(* IEC 61131-3 sources: programs/VI-54/VI-54_20171205/VI-54_20171205/Stations/Screen/LseClass170718/Class/TCPComReceiveData, 1 file *)

(* ---- TCPComReceiveData.st ---- *)
(*!
<Class
	Name               = "TCPComReceiveData"
	Revision           = "1.4"
	RealtimeTask       = "false"
	CyclicTask         = "false"
	BackgroundTask     = "false"
	DefBackground      = "100 ms"
	Sigmatek           = "false"
	OSInterface        = "false"
	HighPriority       = "false"
	Automatic          = "false"
	UpdateMode         = "Prescan"
	SharedCommandTable = "true"
	Objectsize         = "(484,120)"
	Comment            = "this class is used for receiving data from a connected station">
	<Channels>
		<Server Name="Timeout" Visualized="false" Initialize="true" WriteProtected="true" Retentive="false" Comment="Timeout for the receiving process"/>
		<Client Name="coStdLib" Required="false" Internal="false" Comment="object channel to StdLib (don&apos;t connect!)"/>
		<Client Name="coSystemLogging" Required="false" Internal="false" Comment="object channel to SystemLogging (optional)"/>
		<Client Name="CriticalSection" Required="true" Internal="true"/>
	</Channels>
	<Dependencies>
		<Files>
			<File Path=".\Class\TCPComReceiveData\SynchRdWr.h" Include="true"/>
		</Files>
	</Dependencies>
	<RevDoku>
		<Owner Company="Sigmatek"/>
		<Dokumentation Revision="1.4" Date="2016-05-19" Author="GreJoh" Company="Sigmatek" Description="Client coSystemLogging must not be connected."/>
		<Dokumentation Revision="1.3" Date="2015-09-29" Author="BraLis" Company="Sigmatek" Description="insert the method SystemLogging::LogEventText instead of TRACE-Messages"/>
		<Dokumentation Revision="1.2" Date="2015-04-16" Company="Sigmatek"/>
	</RevDoku>
	<Network Name="TCPComReceiveData">
		<!-- List of Components in this network -->
		<Components>
			<Object
				Name       = "_base"
				Class      = "TCPComReceive"
				Position   = "(256,120)"
				Visualized = "false">
				<Channels>
					<Server Name="ClassSvr"/>
					<Server Name="ID_Source"/>
					<Server Name="sRecvCnt"/>
					<Client Name="toDataManager"/>
				</Channels>
			</Object>
			<Object
				Name       = "CriticalSection"
				Class      = "CriticalSection"
				Position   = "(210,540)"
				Visualized = "false">
				<Channels>
					<Server Name="ClassSvr"/>
				</Channels>
			</Object>
		</Components>
		<Comments>
		</Comments>
		<!-- List of Connections in this network -->
		<Connections>
			<Connection Source="this.CriticalSection" Destination="CriticalSection.ClassSvr"/>
			<Connection Source="this.ClassSvr" Destination="_base.ClassSvr" Vertices="(1044,210),(872,210),"/>
			<Connection Source="this.ID_Source" Destination="_base.ID_Source" Vertices="(1044,270),(872,270),"/>
			<Connection Source="this.sRecvCnt" Destination="_base.sRecvCnt" Vertices="(1044,330),(872,330),"/>
			<Connection Source="_base.toDataManager" Destination="this.toDataManager" Vertices="(256,210),(38,210),"/>
		</Connections>
		<!-- Headerfiles -->
		<Options>
		</Options>
	</Network>
</Class>
*)
#pragma using TCPComReceive

TCPComReceiveData : CLASS
: TCPComReceive
	TYPE
	  t_e_SendSteps :
	  (
	    TCPComSend_Idle,
	    TCPComSend_SendData,
	    TCPComSend_WaitAck
	  )$UDINT;
	  t_e_Startup :
	  (
	    Startup_WaitOnline,
	    Startup_GetData,
	    Startup_Send
	  )$UDINT;
#pragma pack(push, 1)
	  t_s_CBCount : STRUCT
	    udSending : DINT;
	    udSended : DINT;
	    udReceived : DINT;
	    udNoReceiverConnected : DINT;
	    udJobDeleted : DINT;
	    udTimeout : DINT;
	    udGlobalReceiveError : DINT;
	  END_STRUCT;
#pragma pack(pop)
#pragma pack(push, 1)
	  t_s_Data : STRUCT
	    udID : UDINT;
	    pValue : ^void;
	    udLength : UDINT;
	  END_STRUCT;
#pragma pack(pop)
#pragma pack(push, 1)
	  t_s_SendData : STRUCT
	    bActive : BOOL;
	    udElements : UDINT;
	    aData : ARRAY [0..SynchRdWr_MaxObjects-1] OF t_s_Data;
	  END_STRUCT;
#pragma pack(pop)
	END_TYPE
  //Servers:
	Timeout 	: SvrCh_UDINT;
  //Clients:
	coStdLib 	: CltChCmd__StdLib;
	CriticalSection 	: CltChCmd_CriticalSection;
	coSystemLogging 	: CltChCmd_SystemLogging;
  //Variables:
		aObjects : ARRAY [0..SynchRdWr_MaxObjects-1] OF ^ReadValue;

		udNumberObjects 	: UDINT;
		udRxCounter 	: UDINT;
		IsCon_coSystemLogging 	: BOOL;
  //Functions:

	FUNCTION VIRTUAL GLOBAL Init;

	FUNCTION VIRTUAL GLOBAL CallBackReceiver
		VAR_INPUT
			DestinationID 	: DINT;
			SourceID 	: DINT;
			size 	: UDINT;
			pdata 	: ^USINT;
		END_VAR
		VAR_OUTPUT
			retcode 	: BOOL;			//! <Variable Comment="TRUE .. erfolgreich Empfangen .._MNG_Recived &#13;&#10;FALSE.. Fehler beim Empfangen .._MNG_GlobalReciveError" Name="CallBackReceiver.retcode"/>
		END_VAR;
				//! <Function Comment="Is used to register a receive object." Name="LoginObject"/>
	FUNCTION GLOBAL LoginObject
		VAR_INPUT
			udID 	: UDINT;			//! <Variable Comment="Unique ID number" Name="LoginObject.udID"/>
			pThis 	: ^ReadValue;			//! <Variable Comment="Thispointer" Name="LoginObject.pThis"/>
		END_VAR
		VAR_OUTPUT
			bSuccessful 	: BOOL;			//! <Variable Comment="TRUE.. Method was successful&#13;&#10;FALSE.. Error" Name="LoginObject.bSuccessful"/>
		END_VAR;
  //Tables:
	FUNCTION @STD
		VAR_OUTPUT
			ret_code	: CONFSTATES;
		END_VAR;
	FUNCTION GLOBAL TAB @CT_;
END_CLASS;

#pragma using CriticalSection
#pragma usingLtd _StdLib
#pragma usingLtd SystemLogging

#pragma usingLtd ReadValue

FUNCTION GLOBAL TCPComReceiveData::LoginObject
	VAR_INPUT
		udID 	: UDINT;
		pThis 	: ^ReadValue;
	END_VAR
	VAR_OUTPUT
		bSuccessful 	: BOOL;
	END_VAR

  // Übergabeparameter auf Grenzen prüfen
  if udID >= sizeof(aObjects) / sizeof(aObjects[0]) then
    if IsCon_coSystemLogging = TRUE then
      coSystemLogging.LogEventText("TCPComReceiveData::LoginObject(): Übergabeparameter usID verletzt die Grenzen");
    end_if;
    bSuccessful := false;
    return;
  end_if;

  // Prüfen ob die ID bereits belegt ist
  if aObjects[udID] <> NIL then
    if IsCon_coSystemLogging = TRUE then
      coSystemLogging.LogEventText("TCPComReceiveData::LoginObject(): Index für Profilpunkt bereits belegt");
    end_if;
    bSuccessful := false;
    return;
  end_if;

  // This-Pointer von RdWr-Object speichern,
  // somit ist dieser Index belegt
  aObjects[udID] := pThis;

  // angemeldete Punkte zählen
  udNumberObjects += 1;

  // Methode war erfolgreich
  bSuccessful := true;

END_FUNCTION

FUNCTION VIRTUAL GLOBAL TCPComReceiveData::CallBackReceiver
	VAR_INPUT
		DestinationID 	: DINT;
		SourceID 	: DINT;
		size 	: UDINT;
		pdata 	: ^USINT;
	END_VAR
	VAR_OUTPUT
		retcode 	: BOOL;
	END_VAR
  VAR
    tmpIndex  : UDINT;
    pObject   : ^ReadValue;
  END_VAR

  // Rückgabewert initialisieren
  Retcode := false;

  // Übergabeparameter prüfen
  if pData = NIL then
    if IsCon_coSystemLogging = TRUE then
      coSystemLogging.LogEventText("TCPComReceiveData::ReceiveData(): Pointer auf Daten ungültig");
    end_if;
    return;
  end_if;

  tmpIndex := pdata^;

  // Index prüfen
  if tmpIndex < sizeof(aObjects) / sizeof(aObjects[0]) then
    //Pointer auf ID holen
    pObject := aObjects[tmpIndex];

    // Prüfen ob Objekt verfügbar
    if pObject <> NIL then

      // Daten weiterleiten
      if pObject^.SetData(pdata, size) = false then
        if IsCon_coSystemLogging = TRUE then
          coSystemLogging.LogEventText("TCPComReceiveData::ReceiveData(): Empfangen der Daten in Indexobjekt fehlgeschlagen");
        end_if;
      end_if;

    else
      if IsCon_coSystemLogging = TRUE then
        coSystemLogging.LogEventText("TCPComReceiveData::ReceiveData(): Index zum Empfangen nicht belegt");
      end_if;
    end_if;

  else
    if IsCon_coSystemLogging = TRUE then
      coSystemLogging.LogEventText("TCPComReceiveData::ReceiveData(): Indexüberlauf eim Empfangen");
    end_if;
  end_if;

  // Empfangene Packete zählen
  udRxCounter += 1;

  // alles korrekt empfangen
  Retcode := true;

END_FUNCTION

FUNCTION VIRTUAL GLOBAL TCPComReceiveData::Init

  TCPComReceive::Init();

  if _FirstScan then

    //-----------------------------------------------------------------------------------------
    //  check client-connnections and set flags
    //-----------------------------------------------------------------------------------------
    if (IsClientConnected(#coSystemLogging)) then
      IsCon_coSystemLogging := TRUE;
    else
      IsCon_coSystemLogging := FALSE;
    end_if;

  end_if;

END_FUNCTION
